Universal Robots PolyScope program: demo str weld.urp

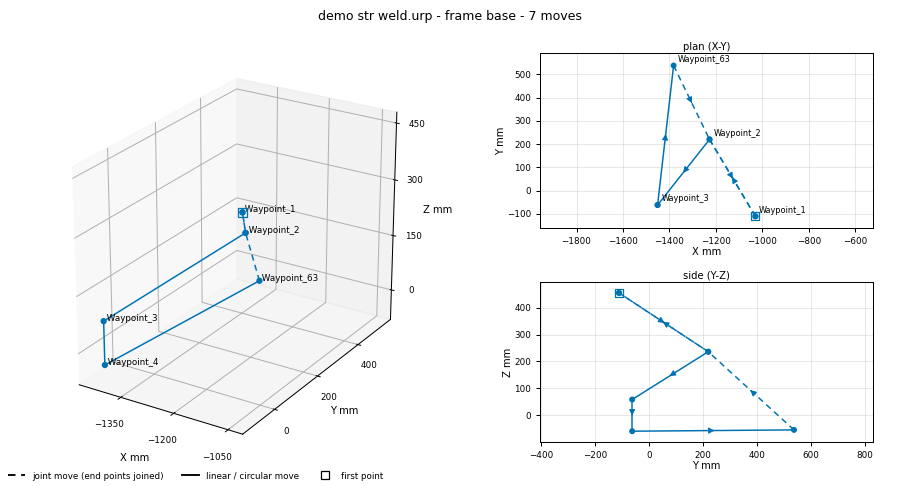
[picture p0: tool path of demo str weld.urp in frame base, 7 of 7 moves have a stored position in this frame; points joined in program order, loops and branches not executed]
Program demo str weld (installation=default directory=/programs createdIn=5.21.3 lastSavedIn=5.21.3 robotSerialNumber=20246801938)
Calibrated DH parameters: a=[-0.000071, -0.790281, -0.600694, 0.000061, -0.000039, 0]; d=[0.236272, 604.465945, 132.116513, -736.382239, 0.159268, 0.154005]; alpha=[1.570254, -0.000567, 0.000559, 1.571709, -1.56999, 0]; deltaTheta=[0, -0.409357, 7.293326, -0.600784, -0.000001, -0.000001]
InitVariablesNode
Robot Program (runOnlyOnce=true)
  Set NoAction tcp=pretend_welder
  MoveJ speed 60 deg/s, acceleration 80 deg/s^2 (useActiveTCP=true optimoveEnabled=false optiMoveSpeed=0.3 optiMoveAcceleration=0.09) feature=Base
    SafeHome (positionOptionType=SPEED_AND_ACCELERATION speed=1.047198 acceleration=1.396263 nextMotionTime=2)
    Waypoint Waypoint_1: TCP in base x=-1030.165 y=-110.755 z=454.213 mm, rx=1.6835 ry=-2.4103 rz=-0.3725 rad; joints [-20.283, -69.554, 90.976, 63.422, -0.136, -102.51] deg; TCP offset x=-9.5 y=-328 z=105.73 mm, rx=1.2092 ry=-1.2092 rz=1.2092 rad
    Waypoint Waypoint_2: TCP in base x=-1227.598 y=220.265 z=236.167 mm, rx=0.2832 ry=3.09 rz=0.0697 rad; joints [-20.205, -68.009, 92.689, -22.783, 80.38, -3.042] deg
    SuppressedNode
      Waypoint Waypoint_59: TCP in base x=-1227.598 y=220.265 z=517.582 mm, rx=0.2832 ry=3.09 rz=0.0697 rad; joints [-20.196, -72.607, 76.22, -1.718, 80.38, -3.031] deg
  MoveL speed 250 mm/s, acceleration 1200 mm/s^2 (useActiveTCP=true optimoveEnabled=false optiMoveSpeed=0.3 optiMoveAcceleration=0.09) feature=Base
    SuppressedNode
      Waypoint Waypoint_7: TCP in base x=-1378.646 y=794.794 z=29.81 mm, rx=0.2832 ry=3.09 rz=0.0697 rad; joints [-40.995, -39.743, 60.872, -18.968, 59.599, -3.836] deg; TCP offset x=-9.5 y=-328 z=105 mm, rx=1.2092 ry=-1.2092 rz=1.2092 rad
    Waypoint Waypoint_3: TCP in base x=-1451.225 y=-61.935 z=58.883 mm, rx=0.1877 ry=3.097 rz=0.0438 rad; joints [-4.252, -49.636, 77.275, -25.571, 92.776, -1.621] deg
    Waypoint Waypoint_4: TCP in base x=-1451.225 y=-61.935 z=-58.667 mm, rx=0.1877 ry=3.097 rz=0.0438 rad; joints [-4.256, -45.514, 80.122, -32.539, 92.773, -1.627] deg
  Folder turn ext on
    URCap WireTank Serial (WireTank Serial, WireTank, LLC) dataModel(NODE_TITLE=Serial Bridge uR1, Command=[252,82,49], QUERY=false, OUTPUT_ENTRY=Static, byte_array=true, Variable(key=OUTPUT_VARIABLE, variable(name=HwResp)))
    URCap WireTank Serial (WireTank Serial, WireTank, LLC) dataModel(NODE_TITLE=Serial Bridge uR1, Command=[252,82,49], byte_array=true, QUERY=false, OUTPUT_ENTRY=Static, Variable(key=OUTPUT_VARIABLE, variable=HwResp))
    Wait Sleep waitTime=1
    SuppressedNode
      Script: turn_extrusion_on()
    Set DigitalOutput pin=digital_out[0]; digitalValue=1
  Wait Sleep waitTime=1
  MoveL speed 10 mm/s, acceleration 1200 mm/s^2 (useActiveTCP=true optimoveEnabled=false optiMoveSpeed=0.3 optiMoveAcceleration=0.09) feature=Base
    Waypoint Waypoint_63: TCP in base x=-1382.264 y=538.31 z=-53.825 mm, rx=0.1877 ry=3.097 rz=0.0438 rad; joints [-32.533, -44.152, 76.93, -30.501, 64.516, -2.709] deg
    SuppressedNode
      Waypoint Waypoint_4: TCP in base x=-1451.225 y=-61.935 z=-58.667 mm, rx=0.1877 ry=3.097 rz=0.0438 rad; joints [-4.256, -45.514, 80.122, -32.539, 92.773, -1.627] deg
    SuppressedNode
      Waypoint Waypoint_6: TCP in base x=-1215.608 y=580.103 z=-51.815 mm, rx=0.1937 ry=3.1132 rz=0.1734 rad; joints [-38.042, -52.199, 93.642, -40.799, 59.177, -6.725] deg
    SuppressedNode
      Waypoint Waypoint_5: TCP in base x=-1209.73 y=609.115 z=-47.444 mm, rx=0.1937 ry=3.1132 rz=0.1734 rad; joints [-39.442, -51.954, 92.704, -40.097, 57.776, -6.743] deg
  URCap WireTank Serial (WireTank Serial, WireTank, LLC) dataModel(QUERY=false, byte_array=true, NODE_TITLE=Serial Bridge uR0, Command=[252,82,48], OUTPUT_ENTRY=Static, Variable(key=OUTPUT_VARIABLE, variable(name=HwResp)))
  MoveL speed 250 mm/s, acceleration 1200 mm/s^2 (useActiveTCP=true optimoveEnabled=false optiMoveSpeed=0.3 optiMoveAcceleration=0.09) feature=Base
    MoveDirectionNode (selectedDirection=ZPlus)
      Until DISTANCE (allowActions=false deceleration=3 distanceNodeType=STOP) Distance=0.15; motionParameters(blendRadius=0)
  Set DigitalOutput pin=digital_out[0]; digitalValue=0
  MoveJ speed 60 deg/s, acceleration 80 deg/s^2 (useActiveTCP=true optimoveEnabled=false optiMoveSpeed=0.3 optiMoveAcceleration=0.09) feature=Base
    Waypoint Waypoint_2: TCP in base x=-1227.598 y=220.265 z=236.167 mm, rx=0.2832 ry=3.09 rz=0.0697 rad; joints [-20.205, -68.009, 92.689, -22.783, 80.38, -3.042] deg; TCP offset x=-9.5 y=-328 z=105.73 mm, rx=1.2092 ry=-1.2092 rz=1.2092 rad
    Waypoint Waypoint_1: TCP in base x=-1030.165 y=-110.755 z=454.213 mm, rx=1.6835 ry=-2.4103 rz=-0.3725 rad; joints [-20.283, -69.554, 90.976, 63.422, -0.136, -102.51] deg
  SafeHome (positionOptionType=SPEED_AND_ACCELERATION speed=1.047198 acceleration=1.396263 nextMotionTime=2)
